DATA_BLOCK "Debug"
{ S7_Optimized_Access := 'TRUE' }
VERSION : 0.1
NON_RETAIN
// ATTRIBUTES
// AUTO_NUMBER = False
// BLOCK_NUMBER = 5
// END_ATTRIBUTES
   VAR
      Bypass : Array[0..100] of Bool;
      Squence : Array[0..100] of Bool;
   END_VAR


BEGIN
   Bypass[3] := 0;

END_DATA_BLOCK

